TYPE FILE_PATH_DATA :
STRUCT
	DRIVE : STRING(3);
	DIRECTORY : STRING(STRING_LENGTH);
	FILENAME : STRING;
END_STRUCT
END_TYPE

(* stored: Version 1.1.0.1, ProductVersion 3.1.4024.4
   DUT FILE_PATH_DATA: Id {1cdd1cda-7d0d-4cdc-bdc3-8ee80cceb3a3} *)
